{attribute 'global_init_slot' := '40500'} // make sure variables are initialized before other GVLs
VAR_GLOBAL

Global_Leak : REAL := 0;
Global_Pressure : REAL := 0.0079;
New_Pressure : REAL := 22.0; //Torr
Global_OverridePressure : BOOL := FALSE;

END_VAR

(* stored: Version 1.1.0.1, ProductVersion 3.1.4022.12
   GVL GVL_Variables: Id {db066f99-a8da-4e2a-bb31-48157f970b30} *)
